Universal Robots PolyScope program: machine_tending_UR.urp

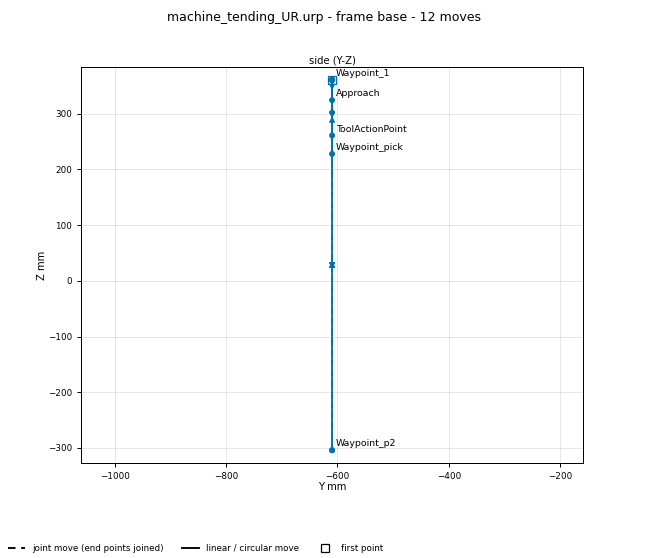
[picture p0: tool path of machine_tending_UR.urp in frame base, 12 of 12 moves have a stored position in this frame; points joined in program order, loops and branches not executed]
Program machine_tending_UR (installation=default directory=/home/ur/ursim-current/programs createdIn=5.14.0 lastSavedIn=5.14.0 robotSerialNumber=20195299999)
Calibrated DH parameters: a=[0, -0.6127, -0.57155, 0, 0, 0]; d=[0.1807, 0, 0, 0.17415, 0.11985, 0.11655]; alpha=[1.570796, 0, 0, 1.570796, -1.570796, 0]; deltaTheta=[0, 0, 0, 0, 0, 0]
InitVariablesNode variables(variable(name=Pallet_1_lct, expression=1), variable(name=Pallet_1_lno, expression=1), variable(name=Pallet_1_sep, expression=False), variable(name=Pallet_1_tct, expression=1), variable(name=pallet_cnt, expression=1))
Robot Program (runOnlyOnce=false)
  Script file /home/ur/ursim-current/programs/machine_tending_init.script
    | # variables
    | task_running = False
    | empty_feeder = True
    | 
    | picking = False
    | loading = False
    | machining = False
    | unloading = False
    | placing = False
    | 
    | cycle_counter = 0
    | 
    | # I/O MAPPING
    | DOOR_OUT = 2
    | CHUCK_OUT = 4
    | CYCLE_OUT = 6
    | 
    | # functions
    | def cycle_completed():
    | 	picking = False
    |     loading = False
    |     machining = False
    |     unloading = False
    |     placing = False
    | end
    | 
    | def get_robot_status():
    |     if task_running:
    |         return "RUNNING"
    |     else:
    |         if empty_feeder:
    |     	    return "READY"
    |         else:
    |             return "COMPLETED"
    |         end
    |     end
    | end
    | 
    | def get_door_status():
    |     if get_standard_digital_out(DOOR_OUT):
    |     	return "OPEN"
    |     else:
    |         return "CLOSE"
    |     end
    | end
    | 
    | def get_chuck_status():
    |     if get_standard_digital_out(CHUCK_OUT):
    |     	return "OPEN"
    |     else:
    |         return "CLOSE"
    |     end
    | end
    | 
    | def get_cycle_status():
    |     if get_standard_digital_out(CYCLE_OUT):
    |     	return "STARTED"
    |     else:
    |         return "STOPPED"
    |     end
    | end
  URCap HMI (Robpod HMI URcap, Robpod Cloud) dataModel(robpod.hmi.selected=/home/ur/ursim-current/programs/machine_tending_hmi.hmi)
  Wait Condition expression=task_running
  Script: empty_feeder =  False
  Loop Counting (count=6) loopVariable(name=Loop_1)
    Folder PICKING
      Script: picking =  True
      MoveJ speed 60 deg/s, acceleration 80 deg/s^2 (useActiveTCP=true) feature=Base
        Waypoint Waypoint_1: motionParameters(nextMotionTime=1); TCP in base x=-189.632 y=-609.684 z=360.813 mm, rx=-0.0012 ry=3.1163 rz=0.0389 rad; joints [-91.713, -91.856, -121.313, -58.303, 91.392, -1.776] deg
      MoveL speed 250 mm/s, acceleration 1200 mm/s^2 (useActiveTCP=true) feature=Base
        Waypoint Waypoint_pick: motionParameters(nextMotionTime=1.5); TCP in base x=-189.632 y=-609.684 z=227.873 mm, rx=-0.0012 ry=3.1163 rz=0.0389 rad; joints [-91.713, -101.794, -127.463, -42.216, 91.392, -1.776] deg; TCP offset x=0 y=0 z=0 mm, rx=0 ry=0 rz=0 rad
      MoveJ speed 60 deg/s, acceleration 80 deg/s^2 (useActiveTCP=true) feature=Base
        Waypoint Waypoint_1: motionParameters(nextMotionTime=1); TCP in base x=-189.632 y=-609.684 z=360.813 mm, rx=-0.0012 ry=3.1163 rz=0.0389 rad; joints [-91.713, -91.856, -121.313, -58.303, 91.392, -1.776] deg
    Folder LOADING
      Script: loading =  True
      Set DigitalOutput pin=digital_out[2]; digitalValue=1
      Set DigitalOutput pin=digital_out[4]; digitalValue=1
      MoveJ speed 60 deg/s, acceleration 80 deg/s^2 (useActiveTCP=true) feature=Base
        Waypoint Waypoint_1: motionParameters(nextMotionTime=1); TCP in base x=-189.632 y=-609.684 z=360.813 mm, rx=-0.0012 ry=3.1163 rz=0.0389 rad; joints [-91.713, -91.856, -121.313, -58.303, 91.392, -1.776] deg
      MoveL speed 250 mm/s, acceleration 1200 mm/s^2 (useActiveTCP=true) feature=Base
        Waypoint Waypoint_p2: motionParameters(nextMotionTime=2); TCP in base x=-189.632 y=-609.684 z=-304.077 mm, rx=-0.0012 ry=3.1163 rz=0.0389 rad; joints [-91.713, -160.888, -117.225, 6.64, 91.392, -1.776] deg; TCP offset x=0 y=0 z=0 mm, rx=0 ry=0 rz=0 rad
      Set DigitalOutput pin=digital_out[4]; digitalValue=0
      MoveJ speed 60 deg/s, acceleration 80 deg/s^2 (useActiveTCP=true) feature=Base
        Waypoint Waypoint_1: motionParameters(nextMotionTime=1); TCP in base x=-189.632 y=-609.684 z=360.813 mm, rx=-0.0012 ry=3.1163 rz=0.0389 rad; joints [-91.713, -91.856, -121.313, -58.303, 91.392, -1.776] deg
      Set DigitalOutput pin=digital_out[2]; digitalValue=0
      Set DigitalOutput pin=digital_out[6]; digitalValue=1
    Folder MACHINING
      Script: machining =  True
      Wait Sleep waitTime=7.5
    Folder UNLOADING
      Script: unloading =  True
      Set DigitalOutput pin=digital_out[6]; digitalValue=0
      Set DigitalOutput pin=digital_out[2]; digitalValue=1
      MoveJ speed 60 deg/s, acceleration 80 deg/s^2 (useActiveTCP=true) feature=Base
        Waypoint Waypoint_1: motionParameters(nextMotionTime=1); TCP in base x=-189.632 y=-609.684 z=360.813 mm, rx=-0.0012 ry=3.1163 rz=0.0389 rad; joints [-91.713, -91.856, -121.313, -58.303, 91.392, -1.776] deg
      MoveL speed 250 mm/s, acceleration 1200 mm/s^2 (useActiveTCP=true) feature=Base
        Waypoint Waypoint_p2: motionParameters(nextMotionTime=2); TCP in base x=-189.632 y=-609.684 z=-304.077 mm, rx=-0.0012 ry=3.1163 rz=0.0389 rad; joints [-91.713, -160.888, -117.225, 6.64, 91.392, -1.776] deg; TCP offset x=0 y=0 z=0 mm, rx=0 ry=0 rz=0 rad
      Set DigitalOutput pin=digital_out[4]; digitalValue=1
      MoveJ speed 60 deg/s, acceleration 80 deg/s^2 (useActiveTCP=true) feature=Base
        Waypoint Waypoint_1: motionParameters(nextMotionTime=1); TCP in base x=-189.632 y=-609.684 z=360.813 mm, rx=-0.0012 ry=3.1163 rz=0.0389 rad; joints [-91.713, -91.856, -121.313, -58.303, 91.392, -1.776] deg
    Folder PLACING
      Script: placing =  True
      URCap Palletizing (polyscope-pallet-impl, Universal Robots) dataModel(palletFeature=Base, isPalletizing=true, Length(key=objectHeight value=0.005 unit=M), Variable(key=name, variable(name=pallet)), Variable(key=globalCountingVariable, variable(name=pallet_cnt, initializeExpression=1)), Variable(key=layerCountingVariable, variable(name=Pallet_1_lct, initializeExpression=1)), Variable(key=layerNumberVariable, variable(name=Pallet_1_lno, initializeExpression=1)), Variable(key=handleSeparatorVariable, variable(name=Pallet_1_sep, initializeExpression=False)), Variable(key=totalCountVariable, variable(name=Pallet_1_tct, initializeExpression=1)), Variable(key=referencePoint, variable(featureName=referencePoint)), Variable(key=separatorPoint, variable(featureName=separatorPoint))); state(isChildrenLocked=true)
        URCap Patterns (polyscope-pallet-impl, Universal Robots) state(isChildrenLocked=true)
          URCap Pattern (polyscope-pallet-impl, Universal Robots) dataModel(UUID=7c668e3c-cb2c-4940-9bf4-0e86e41bf3d3, patternType=GRID, columns=3, rows=2, Variable(key=nameVariable, variable(name=Grid_Pattern_1))); state(isChildrenLocked=true)
            URCap Item (polyscope-pallet-impl, Universal Robots) dataModel(UUID=a5789785-cf2a-4db8-8095-e19286b8aab9, patternType=GRID, index=0, calibrationDeltaTheta=[0.0, 0.0, 0.0, 0.0, 0.0, 0.0], calibrationA=[0.0, -0.6127, -0.57155, 0.0, 0.0, 0.0], calibrationD=[0.1807, 0.0, 0.0, 0.17415, 0.11985, 0.11655], calibrationAlpha=[1.570796327, 0.0, 0.0, 1.570796327, -1.570796327, 0.0], calibrationJointChecksum=[-1, -1, -1, -1, -1, -1], calibrationStatus=0, calibrationValidChecksum=false, baseToFeature=[0.0, 0.0, 0.0, 0.0, 0.0, 0.0], TCPOffset=[1.6653345369377348E-16, 2.220446049250313E-16, 2.7755575615628914E-16, 0.0, 0.0, 0.0], JointPositions(key=jointpositions, JointPosition(key=[1], Angle(key=pos value=-1.6007 unit=RAD)), JointPosition(key=[2], Angle(key=pos value=-1.7271 unit=RAD)), JointPosition(key=[3], Angle(key=pos value=-2.203 unit=RAD)), JointPosition(key=[4], Angle(key=pos value=-0.808 unit=RAD)), JointPosition(key=[5], Angle(key=pos value=1.5951 unit=RAD)), JointPosition(key=[6], Angle(key=pos value=-0.031 unit=RAD))), Variable(key=variable, variable(name=CornerItem_1)))
            URCap Item (polyscope-pallet-impl, Universal Robots) dataModel(UUID=b1cd539b-edfd-41e8-881c-d714e5329cbc, patternType=GRID, index=1, calibrationDeltaTheta=[0.0, 0.0, 0.0, 0.0, 0.0, 0.0], calibrationA=[0.0, -0.6127, -0.57155, 0.0, 0.0, 0.0], calibrationD=[0.1807, 0.0, 0.0, 0.17415, 0.11985, 0.11655], calibrationAlpha=[1.570796327, 0.0, 0.0, 1.570796327, -1.570796327, 0.0], calibrationJointChecksum=[-1, -1, -1, -1, -1, -1], calibrationStatus=0, calibrationValidChecksum=false, baseToFeature=[0.0, 0.0, 0.0, 0.0, 0.0, 0.0], TCPOffset=[1.6653345369377348E-16, 2.220446049250313E-16, 2.7755575615628914E-16, 0.0, 0.0, 0.0], JointPositions(key=jointpositions, JointPosition(key=[1], Angle(key=pos value=-1.6007 unit=RAD)), JointPosition(key=[2], Angle(key=pos value=-1.7271 unit=RAD)), JointPosition(key=[3], Angle(key=pos value=-2.203 unit=RAD)), JointPosition(key=[4], Angle(key=pos value=-0.808 unit=RAD)), JointPosition(key=[5], Angle(key=pos value=1.5951 unit=RAD)), JointPosition(key=[6], Angle(key=pos value=-0.031 unit=RAD))), Variable(key=variable, variable(name=CornerItem_2)))
            URCap Item (polyscope-pallet-impl, Universal Robots) dataModel(UUID=87029a4b-0bc2-46d6-ae58-111d2dcb8d6a, patternType=GRID, index=2, calibrationDeltaTheta=[0.0, 0.0, 0.0, 0.0, 0.0, 0.0], calibrationA=[0.0, -0.6127, -0.57155, 0.0, 0.0, 0.0], calibrationD=[0.1807, 0.0, 0.0, 0.17415, 0.11985, 0.11655], calibrationAlpha=[1.570796327, 0.0, 0.0, 1.570796327, -1.570796327, 0.0], calibrationJointChecksum=[-1, -1, -1, -1, -1, -1], calibrationStatus=0, calibrationValidChecksum=false, baseToFeature=[0.0, 0.0, 0.0, 0.0, 0.0, 0.0], TCPOffset=[1.6653345369377348E-16, 2.220446049250313E-16, 2.7755575615628914E-16, 0.0, 0.0, 0.0], JointPositions(key=jointpositions, JointPosition(key=[1], Angle(key=pos value=-1.6007 unit=RAD)), JointPosition(key=[2], Angle(key=pos value=-1.7271 unit=RAD)), JointPosition(key=[3], Angle(key=pos value=-2.203 unit=RAD)), JointPosition(key=[4], Angle(key=pos value=-0.808 unit=RAD)), JointPosition(key=[5], Angle(key=pos value=1.5951 unit=RAD)), JointPosition(key=[6], Angle(key=pos value=-0.031 unit=RAD))), Variable(key=variable, variable(name=CornerItem_3)))
            URCap Item (polyscope-pallet-impl, Universal Robots) dataModel(UUID=07230cd9-cc65-412c-bb00-1abe7927dd30, patternType=GRID, index=3, calibrationDeltaTheta=[0.0, 0.0, 0.0, 0.0, 0.0, 0.0], calibrationA=[0.0, -0.6127, -0.57155, 0.0, 0.0, 0.0], calibrationD=[0.1807, 0.0, 0.0, 0.17415, 0.11985, 0.11655], calibrationAlpha=[1.570796327, 0.0, 0.0, 1.570796327, -1.570796327, 0.0], calibrationJointChecksum=[-1, -1, -1, -1, -1, -1], calibrationStatus=0, calibrationValidChecksum=false, baseToFeature=[0.0, 0.0, 0.0, 0.0, 0.0, 0.0], TCPOffset=[1.6653345369377348E-16, 2.220446049250313E-16, 2.7755575615628914E-16, 0.0, 0.0, 0.0], JointPositions(key=jointpositions, JointPosition(key=[1], Angle(key=pos value=-1.6007 unit=RAD)), JointPosition(key=[2], Angle(key=pos value=-1.7271 unit=RAD)), JointPosition(key=[3], Angle(key=pos value=-2.203 unit=RAD)), JointPosition(key=[4], Angle(key=pos value=-0.808 unit=RAD)), JointPosition(key=[5], Angle(key=pos value=1.5951 unit=RAD)), JointPosition(key=[6], Angle(key=pos value=-0.031 unit=RAD))), Variable(key=variable, variable(name=CornerItem_4)))
        URCap Layers (polyscope-pallet-impl, Universal Robots) dataModel(separators=[false], selectedPatterns=[7c668e3c-cb2c-4940-9bf4-0e86e41bf3d3])
        URCap At Each Item (polyscope-pallet-impl, Universal Robots) dataModel(selectedPattern=7c668e3c-cb2c-4940-9bf4-0e86e41bf3d3, selectedPosition=a5789785-cf2a-4db8-8095-e19286b8aab9, Approach_calibrationDeltaTheta=[0.0, 0.0, 0.0, 0.0, 0.0, 0.0], Approach_calibrationA=[0.0, -0.6127, -0.57155, 0.0, 0.0, 0.0], Approach_calibrationD=[0.1807, 0.0, 0.0, 0.17415, 0.11985, 0.11655], Approach_calibrationAlpha=[1.570796327, 0.0, 0.0, 1.570796327, -1.570796327, 0.0], Approach_calibrationJointChecksum=[-1, -1, -1, -1, -1, -1], Approach_calibrationStatus=0, Approach_calibrationValidChecksum=false, Approach_baseToFeature=[0.0, 0.0, 0.0, 0.0, 0.0, 0.0], Approach_TCPOffset=[1.6653345369377348E-16, 1.1102230246251565E-16, 3.3306690738754696E-16, 0.0, 0.0, 0.0], Exit_calibrationDeltaTheta=[0.0, 0.0, 0.0, 0.0, 0.0, 0.0], Exit_calibrationA=[0.0, -0.6127, -0.57155, 0.0, 0.0, 0.0], Exit_calibrationD=[0.1807, 0.0, 0.0, 0.17415, 0.11985, 0.11655], Exit_calibrationAlpha=[1.570796327, 0.0, 0.0, 1.570796327, -1.570796327, 0.0], Exit_calibrationJointChecksum=[-1, -1, -1, -1, -1, -1], Exit_calibrationStatus=0, Exit_calibrationValidChecksum=false, Exit_baseToFeature=[0.0, 0.0, 0.0, 0.0, 0.0, 0.0], Exit_TCPOffset=[1.6653345369377348E-16, 0.0, 2.220446049250313E-16, 0.0, 0.0, 0.0], currentWizardState=MANUAL, Pose(key=refBaseToFeature, Position(key=posePosition, Length(key=X value=0 unit=M), Length(key=Y value=0 unit=M), Length(key=Z value=0 unit=M)), Rotation(key=poseRotation, Angle(key=RX value=0 unit=RAD), Angle(key=RY value=0 unit=RAD), Angle(key=RZ value=0 unit=RAD))), Pose(key=refPose, Position(key=posePosition, Length(key=X value=-0.189632 unit=M), Length(key=Y value=-0.609684 unit=M), Length(key=Z value=0.260971 unit=M)), Rotation(key=poseRotation, Angle(key=RX value=-0.001221 unit=RAD), Angle(key=RY value=3.116277 unit=RAD), Angle(key=RZ value=0.038892 unit=RAD))), JointPositions(key=Approach_jointpositions, JointPosition(key=[1], Angle(key=pos value=-1.6007 unit=RAD)), JointPosition(key=[2], Angle(key=pos value=-1.643961 unit=RAD)), JointPosition(key=[3], Angle(key=pos value=-2.152023 unit=RAD)), JointPosition(key=[4], Angle(key=pos value=-0.942116 unit=RAD)), JointPosition(key=[5], Angle(key=pos value=1.5951 unit=RAD)), JointPosition(key=[6], Angle(key=pos value=-0.031 unit=RAD))), JointPositions(key=Exit_jointpositions, JointPosition(key=[1], Angle(key=pos value=-1.6007 unit=RAD)), JointPosition(key=[2], Angle(key=pos value=-1.603196 unit=RAD)), JointPosition(key=[3], Angle(key=pos value=-2.117317 unit=RAD)), JointPosition(key=[4], Angle(key=pos value=-1.017587 unit=RAD)), JointPosition(key=[5], Angle(key=pos value=1.5951 unit=RAD)), JointPosition(key=[6], Angle(key=pos value=-0.031 unit=RAD))))
          URCap Generated Movements (polyscope-pallet-impl, Universal Robots) state(isChildrenLocked=true)
            MoveJ speed 60 deg/s, acceleration 80 deg/s^2 (useActiveTCP=true) feature=referencePoint
              Waypoint Approach: motionParameters(nextMotionTime=0.5); TCP in base x=-189.632 y=-609.684 z=324.313 mm, rx=-0.0012 ry=3.1163 rz=0.0389 rad; joints [-91.713, -94.192, -123.302, -53.979, 91.392, -1.776] deg; TCP offset x=0 y=0 z=0 mm, rx=0 ry=0 rz=0 rad; feature pose in base x=-189.632 y=-609.684 z=260.971 mm, rx=-0.0012 ry=3.1163 rz=0.0389 rad
            MoveL speed 250 mm/s, acceleration 1200 mm/s^2 (useActiveTCP=true) feature(featureName=referencePoint)
              Waypoint ToolActionPoint: motionParameters(nextMotionTime=1); TCP in base x=-189.632 y=-609.684 z=260.971 mm, rx=-0.0012 ry=3.1163 rz=0.0389 rad; joints [-91.713, -98.956, -126.223, -46.295, 91.392, -1.776] deg; TCP offset x=0 y=0 z=0 mm, rx=0 ry=0 rz=0 rad
            Folder Tool action
              Wait Sleep waitTime=0.01
            MoveL speed 250 mm/s, acceleration 1200 mm/s^2 (useActiveTCP=true) feature(featureName=referencePoint)
              Waypoint Exit_1: motionParameters(nextMotionTime=1); TCP in base x=-189.632 y=-609.684 z=360.813 mm, rx=-0.0012 ry=3.1163 rz=0.0389 rad; joints [-91.713, -91.856, -121.313, -58.303, 91.392, -1.776] deg; TCP offset x=0 y=0 z=0 mm, rx=0 ry=0 rz=0 rad
    Script: cycle_counter = cycle_counter + 1
    Script: cycle_completed()
  Script: task_running = False
  Wait Condition expression=empty_feeder
